{attribute 'hide'}
FUNCTION_BLOCK FB_Hidden

END_FUNCTION_BLOCK

(* stored: Version 1.1.0.1
   POU FB_Hidden: Id {11111111-1111-1111-1111-111111111106} *)
